Staubli VAL3: getJointDate.pgx

program getJointDate(string x_sText, jointRx& x_jJoint)
  local string l_sJntDate[6]
  local bool l_bBool
  local pointRx l_pP
begin
  call split(x_sText,",",l_sJntDate)
  if !bMatlab
    l_sJntDate[0]=toNum(l_sJntDate[0],x_jJoint.j1,l_bBool)
    l_sJntDate[1]=toNum(l_sJntDate[1],x_jJoint.j2,l_bBool)
    l_sJntDate[2]=toNum(l_sJntDate[2],x_jJoint.j3,l_bBool)
    l_sJntDate[3]=toNum(l_sJntDate[3],x_jJoint.j4,l_bBool)
    l_sJntDate[4]=toNum(l_sJntDate[4],x_jJoint.j5,l_bBool)
    l_sJntDate[5]=toNum(l_sJntDate[5],x_jJoint.j6,l_bBool)
  else


    //2015.02.05
    //point转为joint
    toNum(l_sJntDate[0],l_pP.trsf.x,l_bBool)
    toNum(l_sJntDate[1],l_pP.trsf.y,l_bBool)
    toNum(l_sJntDate[2],l_pP.trsf.z,l_bBool)
    toNum(l_sJntDate[3],l_pP.trsf.rx,l_bBool)
    toNum(l_sJntDate[4],l_pP.trsf.ry,l_bBool)
    toNum(l_sJntDate[5],l_pP.trsf.rz,l_bBool)
    call NCVetor(fPrdFrame.trsf,l_pP.trsf)
    link(l_pP,fPrdFrame)
    if pointToJoint(tPrdTool,herej(),l_pP,x_jJoint)==false
      logMsg("关节转换出错"+toString(".3",l_pP.trsf.rx)+"  "+toString(".3",l_pP.trsf.ry)+"  "+toString(".3",l_pP.trsf.rz))
      popUpMsg("关节转换出错")
    endIf
  endIf

end
